PROGRAM prgPersistent
VAR
	fbUSV		: FB_WritePersistentData_CX81xx;
	fb_Reboot: NT_Reboot;
	mTest: BOOL;
	ton_liveCount: Ton;
	int_LiveCount: INT;										//{#lynus.ag#()}
END_VAR

fbUSV(
	eSaveModeData:= eUSVSaveMode.eSaveWhenPowerfail, 
	bLoadPersistentDataOk=> , 
	bPowerFailDetect=> , 
	bError=> , 
	bySaveProcess=> , 
	dwStorageLast24h=> , 
	udiErrorCode=> );
	
fb_Reboot (
	netid := '',
	delay := 5,
	start := mTest);
	

ton_liveCount( 	IN := NOT ton_liveCount.Q,
				PT := T#1M);
				
IF ton_liveCount.Q THEN
	int_LiveCount := int_LiveCount+1;	
END_IF

END_PROGRAM

(* stored: Version 1.1.0.1, ProductVersion 3.1.4024.11
   POU prgPersistent: Id {cf2e0bad-677f-4823-a2bf-489f86d455a8}, SpecialFunc None *)
